FUNCTION_BLOCK FB_RecipeParameter IMPLEMENTS I_RecipeParameter
VAR
	sName		: STRING;
	bValue 		: BOOL;
	iValue		: DINT;
	rValue		: REAL;
	sValue		: STRING;
	psFileValue	: POINTER TO STRING;
	eType		: E_VisuCtrlRecipeParameterType;
END_VAR

PROPERTY BitValue : REFERENCE TO BOOL
GET
BitValue REF= bValue;
END_GET
END_PROPERTY

PROPERTY DataType : REFERENCE TO E_VisuCtrlRecipeParameterType
GET
DataType REF= eType;
END_GET
END_PROPERTY

PROPERTY FileValue : REFERENCE TO STRING
GET
FileValue REF= psFileValue^;
END_GET
END_PROPERTY

PROPERTY IntValue : REFERENCE TO DINT
GET
IntValue REF= iValue;
END_GET
END_PROPERTY

METHOD MR_FirstCycle : BOOL
VAR_INPUT
	eType			: E_VisuCtrlRecipeParameterType;
	sName			: STRING;
	pFileValueAdr	: PVOID;
END_VAR
THIS^.eType := eType;
THIS^.sName := sName;
THIS^.psFileValue := pFileValueAdr;
END_METHOD

PROPERTY Name : REFERENCE TO STRING
GET
Name REF= sName;
END_GET
END_PROPERTY

PROPERTY RealValue : REFERENCE TO REAL
GET
RealValue REF= rValue;
END_GET
END_PROPERTY

PROPERTY StringValue : REFERENCE TO STRING
GET
StringValue REF= sValue;
END_GET
END_PROPERTY

END_FUNCTION_BLOCK

(* stored: Version 1.1.0.1, ProductVersion 3.1.4024.9
   POU FB_RecipeParameter: Id {e082d0f9-d5d4-4c12-bf2d-00afc2239cf2}, SpecialFunc None
   Folder FirstCycle: Id {591bd986-d48e-4ffb-b882-334a612af9d7}
   Folder Propierties: Id {f18b81ec-5194-4c23-a83a-74cf026f8428}
   Property BitValue: Id {b9f7b1fb-fd4e-4b06-8bed-a58005160f10}
   Get Get: Id {1d24c466-3720-4e01-b9b0-16aa6e445b7e}
   Property DataType: Id {58bd609c-8a04-4f5d-b1fb-ebe20f674b97}
   Get Get: Id {e1da5f90-dd5e-4e2e-809b-70976115c319}
   Property FileValue: Id {a934ae69-468b-410d-be04-7c1bef3495e5}
   Get Get: Id {f5ed7b22-2144-4338-bd6e-e4f68f1a1575}
   Property IntValue: Id {497bd756-0db9-4148-bef9-67da3241d40d}
   Get Get: Id {35e72dd1-d366-4395-b0f3-96a2431dfd16}
   Method MR_FirstCycle: Id {3d314273-11fd-4775-b281-f96a1489686b}
   Property Name: Id {1270eeca-d19a-4348-abb5-9b62e66d2d2b}
   Get Get: Id {e5e091c7-4e76-4c88-8a6f-e50a2c46a30e}
   Property RealValue: Id {c85a3678-09a3-4cfd-a69c-34ac7817ea7c}
   Get Get: Id {f765ca23-d1ee-46d6-9217-4391b014d7db}
   Property StringValue: Id {9c3b11cf-18c3-409f-ab10-a9ebaeb68312}
   Get Get: Id {2def68dd-7563-4c44-9738-b8a51bfc30b0} *)
